// TwinCAT 3 PLC project PLC1
// ProgramVersion: 3.1.4026.21
// libraries:
//   Tc2_Standard, * (Beckhoff Automation GmbH)
//   Tc2_System, * (Beckhoff Automation GmbH)
//   Tc2_TcpIp, * (Beckhoff Automation GmbH)
//   Tc2_Utilities, * (Beckhoff Automation GmbH)
// project tree:
//   DUTs/ESP/ EspPacketTerminater.TcDUT (not stored), EspPacketHeader.TcDUT, UpdaterEntry.TcDUT
//   DUTs/RtUdp/ IpAdrUnion.TcDUT (not stored)
//   Functions/ BytesToIpv4.TcPOU (not stored), BytesToUint.TcPOU, BytesToUlint.TcPOU (not stored), CalculatePowerConsumption.TcPOU (not stored), HeaderEndianSwap.TcPOU, Ipv4ToBytes.TcPOU, TailEndianSwap.TcPOU (not stored)
//   GVLs/ GVL_Udp.TcGVL (not stored)
//   Interfaces/ ITF_Cyclic.TcIO (not stored), ITF_EspHost.TcIO, ITF_Node.TcIO, ITF_LinkedList.TcIO (not stored), ITF_NodeFactory.TcIO, ITF_UdpConnection.TcIO, ITF_Updater.TcIO, ITF_UpdaterRegistry.TcIO
//   Object/ESP/ EspHost.TcPOU, UpdaterRegistry.TcPOU, Updater_TestPacket.TcPOU
//   Object/Factories/ EspHostFactory.TcPOU (not stored)
//   Object/IO/ RgbController.TcPOU (not stored)
//   Object/Linked List/ List.TcPOU (not stored)
//   Object/UDP/ DataDecoder.TcPOU, UdpRealtimeSocket.TcPOU, UdpWindowsSocket.TcPOU
//   POUs/ Application.TcPOU, EnergyCalculator.TcPOU, MAIN.TcPOU, MessageBuffer.TcPOU, Tests.TcPOU (not stored), Utility.TcPOU
//   Tasks/ Task_4.TcTTO, _aux.TcTTO (not stored)
//   Tests/ EspNodeController.TcPOU (not stored), GVL_Test.TcGVL, TestHarness.TcPOU (not stored), TestNode.TcPOU, TestNodeFactory.TcPOU, Tests_ListAndFactory.TcPOU, Tests_Udp.TcPOU
// real-time tasks:
//   TASK Task 4: cycle T#100us, priority 1, ADS port 350
//   TASK Aux: cycle T#10ms, priority 2, ADS port 351
// I/O:
//   DEVICE Wifi Router
//   DEVICE Rail IO, AmsNetId 5.143.167.204.4.1
//     Term 1 (EK1200) [EK1200-5000 EtherCAT Power supply (2A E-Bus)]
//       Term 2 (EL9227-5500) [EL9227-5500 Overcurrent protection 24V DC, 2Ch., max. 10A (sum), adjustable, extended functionalities]
//       Term 3 (EL2088) [EL2088 8Ch. Dig. Output 24V, 0.5A, switching to negative]
//       Term 4 (EL9011) [EL9011 End Terminal]
// variable links:
//   PLC1/PLC1 Instance <-> Rail IO/Term 1 (EK1200)/Term 2 (EL9227-5500)
//     Aux Inputs/Utility.EL9227Ch2.MDP5001_922_Input/MDP5001_922_Current <-> OCP Inputs Channel 2/Current
//     Aux Inputs/Utility.EL9227Ch2.MDP5001_922_Input/MDP5001_922_Load <-> OCP Inputs Channel 2/Load
//     Aux Inputs/Utility.EL9227Ch2.MDP5001_922_Input/MDP5001_922_Status <-> OCP Inputs Channel 2/Status
//     Aux Inputs/Utility.EL9227Ch2.MDP5001_922_Input/MDP5001_922_Voltage_In <-> OCP Inputs Channel 2/Voltage In
//     Aux Inputs/Utility.EL9227Ch2.MDP5001_922_Input/MDP5001_922_Voltage_Out <-> OCP Inputs Channel 2/Voltage Out
//     Aux Outputs/Utility.EL9227Ch2.MDP5001_922_Output/MDP5001_922_Control <-> OCP Outputs Channel 2/Control
//     Task_4 Inputs/Utility.EL9227Ch1.MDP5001_922_Input/MDP5001_922_Current <-> OCP Inputs Channel 1/Current
//     Task_4 Inputs/Utility.EL9227Ch1.MDP5001_922_Input/MDP5001_922_Load <-> OCP Inputs Channel 1/Load
//     Task_4 Inputs/Utility.EL9227Ch1.MDP5001_922_Input/MDP5001_922_Status <-> OCP Inputs Channel 1/Status
//     Task_4 Inputs/Utility.EL9227Ch1.MDP5001_922_Input/MDP5001_922_Voltage_In <-> OCP Inputs Channel 1/Voltage In
//     Task_4 Inputs/Utility.EL9227Ch1.MDP5001_922_Input/MDP5001_922_Voltage_Out <-> OCP Inputs Channel 1/Voltage Out
//     Task_4 Outputs/Utility.EL9227Ch1.MDP5001_922_Output/MDP5001_922_Control <-> OCP Outputs Channel 1/Control
//   PLC1/PLC1 Instance <-> Rail IO/Term 1 (EK1200)/Term 3 (EL2088)
//     Task_4 Outputs/Utility.LedStrip._Blue <-> Channel 5/Output
//     Task_4 Outputs/Utility.LedStrip._Green <-> Channel 3/Output
//     Task_4 Outputs/Utility.LedStrip._Red <-> Channel 1/Output

CONFIGURATION PLC1
    RESOURCE PLC ON TwinCAT3
        TASK Task_4(INTERVAL := T#200us, PRIORITY := 1);
        PROGRAM MAIN WITH Task_4 : MAIN;
    END_RESOURCE
END_CONFIGURATION

// ---- DUTs/ESP/EspPacketHeader.TcDUT
TYPE EspPacketHeader :
STRUCT
	StartDelimiter			: UINT := 693;
	PayloadSize				: UINT;
	Reserved1				: ARRAY [1..4] OF BYTE;
	SlaveUid				: ULINT;
	MessageCounter			: ULINT;
	SendersTimestamp		: ULINT;
	TimeDifference			: UDINT;
	NumberOfChainedSLaves	: BYTE;
	EspType					: BYTE;
	Flags					: BYTE;
	HeaderVersion			: BYTE;
	NetworkId				: BYTE;
	ChainDistance			: BYTE;
	JumpsToLive				: BYTE;
	Reserved2				: BYTE;
	CRC32					: UDINT;
END_STRUCT
END_TYPE

// ---- DUTs/ESP/UpdaterEntry.TcDUT
TYPE UpdaterEntry :
STRUCT
	TypeID	: BYTE;
	Version	: BYTE;
	Updater	: ITF_Updater;
END_STRUCT
END_TYPE

// ---- Tests/GVL_Test.TcGVL
{attribute 'qualified_only'}
VAR_GLOBAL
	
END_VAR

// ---- Interfaces/ITF_EspHost.TcIO
INTERFACE ITF_EspHost

METHOD CyclicUpdate : BOOL
VAR_INPUT
END_VAR
END_METHOD

METHOD GetDataBuffer : BOOL
VAR_INPUT
	Address	: REFERENCE TO PVOID;
	Size	: REFERENCE TO UDINT;
END_VAR
END_METHOD

METHOD GetMetadata : EspPacketHeader
VAR_INPUT
END_VAR
END_METHOD

METHOD GetPacketToSend : BOOL
VAR_INPUT
	Address	: REFERENCE TO PVOID;
	Size	: REFERENCE TO UDINT;
END_VAR
END_METHOD

METHOD SetEspType : BOOL
VAR_INPUT
	EspType	: BYTE;
END_VAR
END_METHOD

METHOD SetUID : BOOL
VAR_INPUT
	UID	: ULINT;
END_VAR
END_METHOD

METHOD UpdateMetadata : BOOL
VAR_INPUT
	Data	: EspPacketHeader;
END_VAR
END_METHOD

END_INTERFACE

// ---- Interfaces/ITF_Node.TcIO
INTERFACE ITF_Node

METHOD GetLastNode : ITF_Node
VAR_INPUT
END_VAR
END_METHOD

METHOD GetMyPointer : PVOID
END_METHOD

METHOD GetNextNode : ITF_Node
VAR_INPUT
END_VAR
END_METHOD

METHOD GetPositionInList : UINT
VAR_INPUT
END_VAR
END_METHOD

METHOD SetLastNode : BOOL
VAR_INPUT
	Node	: ITF_Node;
END_VAR
END_METHOD

METHOD SetNextNode : BOOL
VAR_INPUT
	Node	: ITF_Node;
END_VAR
END_METHOD

METHOD SetPositionInList : BOOL
VAR_INPUT
	Index		: UINT;
END_VAR
END_METHOD

END_INTERFACE

// ---- Interfaces/ITF_NodeFactory.TcIO
INTERFACE ITF_NodeFactory

METHOD CreateNode : ITF_Node
VAR_INPUT
END_VAR
END_METHOD

METHOD DestroyNode : BOOL
VAR_INPUT
	Ptr		: PVOID;
END_VAR
END_METHOD

METHOD DoesCreateEqualDestroy : BOOL
END_METHOD

END_INTERFACE

// ---- Interfaces/ITF_UdpConnection.TcIO
INTERFACE ITF_UdpConnection EXTENDS ITF_Cyclic

METHOD IsConnected : BOOL
VAR_INPUT
END_VAR
END_METHOD

METHOD IsSending : BOOL
VAR_INPUT
END_VAR
END_METHOD

PROPERTY LastReceivedIp : T_IPv4Addr
GET
END_GET
END_PROPERTY

PROPERTY ReceiveBufferReference : REFERENCE TO ARRAY [0..TCPADS_MAXUDP_BUFFSIZE - 1] OF BYTE;
GET
END_GET
END_PROPERTY

METHOD TryCloseConnection : HRESULT
VAR_INPUT
END_VAR
END_METHOD

METHOD TryOpenConnection : HRESULT
VAR_INPUT
END_VAR
END_METHOD

METHOD TryReadReceiveBuffer : HRESULT
VAR_INPUT
	DataBuffer		: REFERENCE TO ARRAY [0..TCPADS_MAXUDP_BUFFSIZE - 1] OF BYTE;
END_VAR
END_METHOD

METHOD TrySendData : HRESULT
VAR_INPUT
	IpAddress		: T_IPv4Addr;
	Port			: UDINT;
	DataAddress		: PVOID;
	DataLength		: UDINT;
END_VAR
END_METHOD

END_INTERFACE

// ---- Interfaces/ITF_Updater.TcIO
INTERFACE ITF_Updater

METHOD GetTypeID : BYTE
VAR_INPUT
END_VAR
END_METHOD

METHOD GetVersion : BYTE
VAR_INPUT
END_VAR
END_METHOD

METHOD TryApplyPayload : HRESULT
VAR_INPUT
	PacketAddress	: PVOID;
	PacketLength	: UINT;
	EspHost			: ITF_EspHost;
END_VAR
END_METHOD

METHOD TryGetContents : HRESULT
VAR_INPUT
	Host	: ITF_EspHost;
	Content	: REFERENCE TO STRING(1024);
END_VAR
END_METHOD

METHOD TrySendInstruction : HRESULT
VAR_INPUT
END_VAR
END_METHOD

END_INTERFACE

// ---- Interfaces/ITF_UpdaterRegistry.TcIO
INTERFACE ITF_UpdaterRegistry

METHOD Reset : BOOL
VAR_INPUT
END_VAR
END_METHOD

METHOD ResolveUpdater : ITF_Updater
VAR_INPUT
	TypeID	: BYTE;
	Version	: BYTE;
END_VAR
END_METHOD

METHOD TryRegister : HRESULT
VAR_INPUT
	Updater	: ITF_Updater;
END_VAR
END_METHOD

END_INTERFACE

// ---- POUs/MAIN.TcPOU
PROGRAM MAIN
VAR
	Test	: BOOL := FALSE;
	i		: INT;
END_VAR


i := i + 1;


IF Test THEN
	
	Tests();
	
ELSE
	
	Application();
	
END_IF

END_PROGRAM

// ---- POUs/Application.TcPOU
PROGRAM Application
VAR CONSTANT
	Port 					: UDINT := 10050;
END_VAR
VAR
	UdpWin10				: UdpWindowsSocket('192.168.137.1', Port);
	UdpRt					: UdpRealtimeSocket(Port);
	Udp						: ITF_UdpConnection := UdpRt;
	
	EspFactory				: EspHostFactory;
	List					: List(EspFactory);
	
	DataDecoder				: DataDecoder(Udp, List);
	UpdaterRegistry			: UpdaterRegistry;
	TestUpdater				: Updater_TestPacket;
	
	Init					: BOOL := FALSE;
	i						: BYTE;
	j						: UINT;
	State					: BYTE;
	hr						: HRESULT;

	ReceivedIP				: T_IPv4Addr;
	InputHeader				: EspPacketHeader;	
	TempEspPtr				: POINTER TO EspHost;
	TempEsp					: ITF_EspHost;
	TempEspHeader			: EspPacketHeader;
	
	PacketToSendAdr			: PVOID;
	PacketToSendLength		: UDINT;
	
	ReceivedPacketType		: BYTE;
	ReceivedPacketAddress	: PVOID;
	ReceivedPacketLength	: UINT;
	ReceivedDataLength		: UINT;
	
	PacketsProcessed		: ULINT;
END_VAR


IF NOT Init THEN

	IF Udp.TryOpenConnection() <> S_OK THEN
		
		RETURN;
	
	END_IF

	UpdaterRegistry.TryRegister(TestUpdater);
	
	Init := TRUE;

END_IF





// Multiple processing calls per cycle are possible

FOR i := 0 TO 9 BY 1 DO
	
	Udp.CyclicUpdate();
	
	CASE State OF
		
		0:	// Is data available
			
			hr := DataDecoder.TryFindPacketInBuffer(ReceivedPacketType, ReceivedPacketAddress, ReceivedPacketLength, ReceivedDataLength);
			
			IF hr = S_OK THEN
				
				ReceivedIP := UdpRt.LastReceivedIp;
				
				State := 1;
				
			ELSIF hr <> S_PENDING THEN
				
				EXIT;
				
			END_IF
			
	

		1:	// Decode header
		
			InputHeader := DataDecoder.GetPacketHeader();

			IF InputHeader.SlaveUid = 0 THEN
				
				// Clear buffer
				
				State := 0;
				
			END_IF
			
			State := 2;



		2:	// Check CRC
		
			// CRC Check Function on TargetHeader
			
			// If fail, clear buffer, state := 0
			
			State := 3;



		3:	// Find UID in list
		
			IF List.GetListLength() = 0 THEN
				
				State := 4;
				
			END_IF
		
			FOR j := 1 TO List.GetListLength() BY 1 DO
			
				TempEspPtr := List.GetNode(j).GetMyPointer();
				
				IF TempEspPtr = 0 THEN
					
					// No matching device in list, create
					
					State := 4;
					
				ELSE
					
					// Check if correct UID
					
					TempEsp := TempEspPtr^;
				
					TempEspHeader := TempEsp.GetMetadata();
					
					IF InputHeader.SlaveUid = TempEspHeader.SlaveUid THEN
						
						State := 5;
						
						EXIT;
						
					END_IF
					
				END_IF
				
			END_FOR	
			
			IF j = List.GetListLength() + 1 THEN
				
				State := 4;
				
			END_IF
			
			
			
		4:	// Create device in list
			
			IF List.CreateNode() THEN
						
				TempEspPtr := List.GetNode(List.GetListLength()).GetMyPointer();
				
				TempEsp := TempEspPtr^;
				
				TempEsp.SetUID(InputHeader.SlaveUid);
				
				TempEsp.SetEspType(ReceivedPacketType);
				
				State := 5;
			
			END_IF
			
			
			
		5:	// Apply data
		
			IF TempEsp.UpdateMetadata(InputHeader) THEN
				
				IF TempEsp.GetPacketToSend(PacketToSendAdr, PacketToSendLength) THEN
					
					TempEsp.CyclicUpdate();
					
					State := 6;

				ELSE
					
					State := 7;
	
				END_IF
				
			END_IF
		
		
		
		6:	// Send data
		
			hr := UdpRt.TrySendData(ReceivedIP, Port, PacketToSendAdr, PacketToSendLength);
			
			IF hr <> S_PENDING AND SUCCEEDED(hr) THEN
				
				State := 7;
				
			ELSIF FAILED(hr) THEN
				
				State := 8;
				
			END_IF
		
		
		
		7:	// System function OK
			
			ReceivedIP := '';
			MEMSET(ADR(InputHeader), 0, 48);
			TempEspPtr := 0;
			TempEsp := 0;
			MEMSET(ADR(TempEspHeader), 0, 48);
			DataDecoder.ClearBufferAtLocation(ReceivedPacketAddress, ReceivedPacketLength);
			
			PacketsProcessed := PacketsProcessed + 1;
			State := 0;
			
			
		
		
		8:	// System RX OK, TX FAIL
		
// 		
// 		
// 		
// 		5:
// 		
// 			hr := TempUpdater.TryApplyPayload(ReceivedPacketAddress, ReceivedPacketLength, TempEsp);
// 			
// 			IF hr <> S_PENDING AND SUCCEEDED(hr) THEN
// 				
// 				TempEsp.UpdateMetadata(DataDecoder.CreateMetadataUpdate());
// 				
// 				DataDecoder.ClearBufferAtLocation(ReceivedPacketAddress, ReceivedPacketLength);
// 				
// 				ReceivedPacketAddress := 0;
// 				ReceivedPacketLength := 0;
// 				ReceivedPacketType := 0;
// 			
// 				TargetEspUID := 0;
// 				TempEspPtr := 0;	
// 				TempEsp := 0;
// 				MEMSET(ADR(TempEspHeader), 0, SIZEOF(TempEspHeader));
// 				TempUpdater := 0;
// 				
// 				State := 0;
// 				
// 			END_IF
// 		
// 		
// 			
// 			
// 		1:
// 		
// 			TempUpdater := UpdaterRegistry.ResolveUpdater(ReceivedPacketType, 1);
// 			
// 			IF TempUpdater = 0 THEN
// 				
// 				;// ERROR
// 				
// 			END_IF
// 			
// 			State := 2;
// 			
// 		
// 		
// 		2:
// 		
// 			TargetEspUID := DataDecoder.GetPacketUID();
// 			
// 			IF TargetEspUID = 0 THEN
// 				
// 				;// ERROR
// 				
// 			END_IF
// 			
// 			State := 3;
// 			
// 			
// 			
// 		3:
// 		
// 			FOR j := 1 TO List.GetListLength() BY 1 DO
// 			
// 				TempEspPtr := List.GetNode(j).GetMyPointer();
// 			
// 				TempEsp := TempEspPtr^;
// 				
// 				TempEspHeader := TempEsp.GetMetadata();
// 				
// 				IF TargetEspUID = TempEspHeader.SlaveUid THEN
// 					
// 					FoundEsp := TRUE;
// 					
// 					EXIT;
// 					
// 				END_IF
// 				
// 			END_FOR
// 			
// 			IF FoundEsp THEN
// 				
// 				FoundEsp := FALSE;
// 				
// 				State := 5;
// 				
// 			ELSE
// 				
// 				State := 4;
// 				
// 			END_IF
// 			
// 			
// 			
// 		4:
// 			
// 			IF List.CreateNode() THEN
// 						
// 				TempEspPtr := List.GetNode(List.GetListLength()).GetMyPointer();
// 				
// 				TempEsp := TempEspPtr^;
// 				
// 				TempEsp.SetUID(TargetEspUID);
// 				
// 				TempEsp.SetEspType(ReceivedPacketType);
// 				
// 				State := 5;
// 			
// 			END_IF
// 		
// 		
// 		
// 		5:
// 		
// 			hr := TempUpdater.TryApplyPayload(ReceivedPacketAddress, ReceivedPacketLength, TempEsp);
// 			
// 			IF hr <> S_PENDING AND SUCCEEDED(hr) THEN
// 				
// 				TempEsp.UpdateMetadata(DataDecoder.CreateMetadataUpdate());
// 				
// 				DataDecoder.ClearBufferAtLocation(ReceivedPacketAddress, ReceivedPacketLength);
// 				
// 				ReceivedPacketAddress := 0;
// 				ReceivedPacketLength := 0;
// 				ReceivedPacketType := 0;
// 			
// 				TargetEspUID := 0;
// 				TempEspPtr := 0;	
// 				TempEsp := 0;
// 				MEMSET(ADR(TempEspHeader), 0, SIZEOF(TempEspHeader));
// 				TempUpdater := 0;
// 				
// 				State := 0;
// 				
// 			END_IF
			
	END_CASE

END_FOR

END_PROGRAM

// ---- Object/UDP/UdpWindowsSocket.TcPOU
FUNCTION_BLOCK UdpWindowsSocket IMPLEMENTS ITF_UdpConnection
VAR
	IpAddress			: T_IPv4Addr;
	Port				: UDINT;
	ReceiveBuffer		: ARRAY [0..TCPADS_MAXUDP_BUFFSIZE - 1] OF BYTE;
	
	OpenSocket			: FB_SocketUdpCreate;
	Receive				: FB_SocketUdpReceiveFrom;
	Send				: FB_SocketUdpSendTo;
	SendState			: BYTE;
	Sending 			: BOOL;
	PacketsSent			: ULINT;
	CloseSocket			: FB_SocketClose;
	
	IsConnectionOpen	: BOOL;
END_VAR

METHOD CyclicUpdate : BOOL
VAR
	i	: BYTE;
END_VAR
OpenSocket
(
	sSrvNetId 	:= '', 
	sLocalHost	:= IpAddress, 
	nLocalPort	:= Port, 
);

Send
(
	sSrvNetId	:= '', 
	hSocket		:= OpenSocket.hSocket, 
);

FOR i := 0 TO 9 BY 1 DO
	
	Receive
	(
		sSrvNetId	:= '', 
		hSocket		:= OpenSocket.hSocket, 
		cbLen		:= SIZEOF(ReceiveBuffer), 
		pDest		:= ADR(ReceiveBuffer) 
	);
	
	IF IsSending() OR NOT IsConnectionOpen THEN
	
		Receive(bExecute := FALSE);
		
	ELSE
		
		Receive(bExecute := NOT(Receive.bExecute));
	
	END_IF

END_FOR


CloseSocket
(
	sSrvNetId	:= '', 
	hSocket		:= OpenSocket.hSocket, 
);

IF OpenSocket.hSocket.handle <> 0 AND OpenSocket.bExecute THEN
	
	IsConnectionOpen := TRUE;
	
ELSE

	IsConnectionOpen := FALSE;

END_IF
END_METHOD

//FB_Exit must be implemented explicitly. If there is an implementation, then the
//method is called before the controller removes the code of the function block instance
//(implicit call). The return value is not evaluated.
METHOD FB_Exit: BOOL
VAR_INPUT
    bInCopyCode: BOOL;  // TRUE: the exit method is called in order to leave the instance which will be copied afterwards (online change).  
END_VAR
TryCloseConnection();
END_METHOD

//FB_Init is always available implicitly and it is used primarily for initialization.
//The return value is not evaluated. For a specific influence, you can also declare the
//methods explicitly and provide additional code there with the standard initialization
//code. You can evaluate the return value.
METHOD FB_Init: BOOL
VAR_INPUT
    bInitRetains: BOOL; // TRUE: the retain variables are initialized (reset warm / reset cold)
    bInCopyCode: BOOL;  // TRUE: the instance will be copied to the copy code afterward (online change) 
	IpAddress	: T_IPv4Addr;
	Port		: UDINT;  
END_VAR
THIS^.IpAddress := IpAddress;
THIS^.Port := Port;
END_METHOD

METHOD IsConnected : BOOL
IsConnected := IsConnectionOpen;

RETURN;
END_METHOD

METHOD IsSending : BOOL
IsSending := Sending;

RETURN;
END_METHOD

{warning 'Add property implementation'}
PROPERTY LastReceivedIp : T_IPv4Addr
GET
LastReceivedIp := Receive.sRemoteHost;
END_GET
END_PROPERTY

{warning 'Add property implementation'}
PROPERTY LastReceivedPort : UDINT
GET
LastReceivedPort := Receive.nRemotePort;
END_GET
END_PROPERTY

{warning 'Add property implementation'}
PROPERTY ReceiveBufferReference : REFERENCE TO ARRAY [0..(TCPADS_MAXUDP_BUFFSIZE - 1)] OF BYTE
GET
ReceiveBufferReference REF= ReceiveBuffer;
END_GET
END_PROPERTY

METHOD TryCloseConnection : HRESULT
TryCloseConnection := S_PENDING;

OpenSocket(bExecute := FALSE);

CloseSocket(bExecute := TRUE);

IF OpenSocket.hSocket.handle = 0 THEN
	
	TryCloseConnection := S_OK;

ELSIF OpenSocket.bError THEN

	TryCloseConnection := -1;	

END_IF

RETURN;
END_METHOD

METHOD TryOpenConnection : HRESULT
TryOpenConnection := S_PENDING;

CloseSocket(bExecute := FALSE);

OpenSocket(bExecute := TRUE);

IF OpenSocket.hSocket.handle <> 0 THEN
	
	TryOpenConnection := S_OK;

ELSIF OpenSocket.bError THEN

	TryOpenConnection := -1;	

END_IF

RETURN;
END_METHOD

METHOD TryReadReceiveBuffer : HRESULT
VAR_INPUT
	DataBuffer		: REFERENCE TO ARRAY [0..TCPADS_MAXUDP_BUFFSIZE - 1] OF BYTE;
END_VAR
VAR
	i				: UDINT;
END_VAR
TryReadReceiveBuffer := S_PENDING;

IF ReceiveBuffer[0] = 0 THEN
	
	TryReadReceiveBuffer := -1;

	RETURN;	

END_IF

FOR i := 0 TO TCPADS_MAXUDP_BUFFSIZE BY 1 DO
	
	IF ReceiveBuffer[i] = 0 THEN
		
		EXIT;
		
	END_IF

	DataBuffer[i] := ReceiveBuffer[i];

END_FOR

IF ReceiveBuffer[0] <> 0 THEN
	
	TryReadReceiveBuffer := S_OK;

ELSE

	TryReadReceiveBuffer := -2;

END_IF

RETURN;
END_METHOD

METHOD TrySendData : HRESULT
VAR_INPUT
	IpAddress		: T_IPv4Addr;
	Port			: UDINT;
	DataAddress		: PVOID;
	DataLength		: UDINT;
END_VAR
TrySendData := S_PENDING;

IF NOT IsConnected() THEN
	
	TrySendData := -1;
	
	RETURN;

END_IF

Send
(
	sRemoteHost	:= IpAddress, 
	nRemotePort	:= Port, 
	cbLen		:= DataLength, 
	pSrc		:= DataAddress, 
	bExecute	:= TRUE, 
);

Sending := TRUE;

CASE SendState OF
	
	0:
	
		IF Send.bBusy THEN
			
			SendState := 1;
			
		END_IF



	1:
	
		IF Send.bError THEN
			
			Send(bExecute := FALSE);
			
			TrySendData := -1;
			
			SendState := 0;
			
			Sending := FALSE;
			
			RETURN;
		
		ELSIF NOT Send.bBusy THEN
			
			Send(bExecute := FALSE);
		
			TrySendData := S_OK;
			
			PacketsSent := PacketsSent + 1;
			
			SendState := 0;
			
			Sending := FALSE;
			
			RETURN;
		
		END_IF
END_CASE
END_METHOD

END_FUNCTION_BLOCK

// ---- Object/UDP/UdpRealtimeSocket.TcPOU
{attribute 'c++_compatible'}
FUNCTION_BLOCK UdpRealtimeSocket IMPLEMENTS ITcIoUdpProtocolRecv, ITF_UdpConnection
VAR
	{attribute 'TcInitSymbol'}
	_ObjectId				: OTCID; 
	_ipUdp					: ITcIoUdpProtocol;
	_UdpPort				: UINT := 10000;
	_ReceivedPackets		: ULINT;
	_LastReceivedIpAddr 	: IpAdrUnion;
	_LastReceivedPort		: UDINT; 
	_LastSentIpAddr			: IpAdrUnion;
	_hrInit 				: HRESULT;
	_SocketOpen				: BOOL;
	_Sending				: BOOL;
	
	_ReceivedData			: PVOID;
	_ReceivedDataLength		: UDINT;
		
	_ReceiveBuffer			: ARRAY [0..TCPADS_MAXUDP_BUFFSIZE - 1] OF BYTE;

END_VAR

METHOD CyclicUpdate : BOOL
IF _ipUdp <> 0 THEN
	
	_ipUdp.CheckReceived();
	
END_IF

IF _ReceivedData <> 0 THEN

	MEMCPY(ADR(_ReceiveBuffer), _ReceivedData, _ReceivedDataLength);
	
	_ReceivedData := 0;
	
	_ReceivedDataLength := 0;

END_IF
END_METHOD

METHOD FB_exit : BOOL
VAR_INPUT
	bInCopyCode : BOOL; // if TRUE, the exit method is called for exiting an instance that is copied afterwards (online change).
END_VAR
IF (NOT bInCopyCode AND _ipUdp <> 0) THEN //Shutdown
	_ipUdp.UnregisterReceiver(_UdpPort);
	FW_SafeRelease(ADR(_ipUdp));
	_SocketOpen := FALSE;
	FB_exit := TRUE;
ELSE
	FB_exit := FALSE;
END_IF
END_METHOD

METHOD FB_init : BOOL
VAR_INPUT
	bInitRetains : BOOL; // if TRUE, the retain variables are initialized (warm start / cold start)
	bInCopyCode : BOOL;  // if TRUE, the instance afterwards gets moved into the copy code (online change)
	Port	: UDINT;
END_VAR
VAR
	//ipSrv: ITComObjectServer;
END_VAR
_UdpPort := TO_UINT(Port);
// 
// IF NOT bInCopyCode THEN // no online change
// 	IF ipUdp = 0 AND ObjectId <> 0 THEN
// 	 hrInit := FW_ObjMgr_GetObjectInstance(oid:=ObjectId, iid:=TC_GLOBAL_IID_LIST.IID_ITcIoUdpProtocol, pipUnk:=ADR(ipUdp) );
// 		IF SUCCEEDED(hrInit) THEN 
// 			IF SUCCEEDED(ipUdp.RegisterReceiver(UdpPort, THIS^)) THEN //open port
// 				SocketOpen := TRUE;
// 				FB_init := TRUE;
// 			ELSE 
// 				FB_init := FALSE; 
// 				FW_SafeRelease(ADR(ipUdp));
// 			END_IF
// 		END_IF
// 	ELSIF ObjectId = 0 THEN 
// 		FB_init := FALSE; 
// 		hrInit := ERR_INVALID_PARAM; 				
// 	END_IF
// END_IF
END_METHOD

METHOD FB_reinit : BOOL
VAR_INPUT
END_VAR
IF (_ipUdp <> 0) THEN 
  _ipUdp.RegisterReceiver(_UdpPort, THIS^);
  _SocketOpen := TRUE;
  FB_reinit := TRUE; 
END_IF
END_METHOD

METHOD IsConnected : BOOL
IsConnected := _SocketOpen;

RETURN;
END_METHOD

METHOD IsSending : BOOL
IsSending := _Sending;

RETURN;
END_METHOD

PROPERTY LastReceivedIp : T_IPv4Addr
GET
LastReceivedIp := BytesToIpv4(_LastReceivedIpAddr.IpByte);
END_GET
END_PROPERTY

{warning 'Add property implementation'}
PROPERTY LastReceivedPort : UDINT
GET
LastReceivedPort := _LastReceivedPort;
END_GET
END_PROPERTY

{warning 'Add property implementation'}
PROPERTY ReceiveBufferReference : REFERENCE TO ARRAY [0..(TCPADS_MAXUDP_BUFFSIZE - 1)] OF BYTE
GET
ReceiveBufferReference REF= _ReceiveBuffer;
END_GET
END_PROPERTY

{attribute 'object_name' := 'ReceiveData'}
{attribute 'c++_compatible'}
{attribute 'pack_mode' := '4'}
{attribute 'show'}
{attribute 'minimal_input_size' := '4'}
METHOD ReceiveData : HRESULT
VAR_INPUT
	ipAddr	: UDINT;
	udpDestPort	: UINT;
	udpSrcPort	: UINT;
	nData	: UDINT;
	pData	: PVOID;
	pVlan	: POINTER TO ETYPE_VLAN_HEADER := 0;
END_VAR
_ReceivedPackets := _ReceivedPackets + 1;

_LastReceivedIpAddr.IpUdint := ipAddr;

_LastReceivedPort := TO_UDINT(udpDestPort);

IF _ipUdp <> 0 THEN
	
	//ipUdp.SendData(ipAddr, udpSrcPort, udpDestPort, nData, pData, TRUE, 0); // send data back

	_ReceivedData := pData;
	
	_ReceivedDataLength := nData;
	
END_IF
END_METHOD

{attribute 'object_name' := 'TcAddRef'}
{attribute 'c++_compatible'}
{attribute 'pack_mode' := '4'}
{attribute 'show'}
{attribute 'minimal_input_size' := '4'}
METHOD TcAddRef : UDINT
END_METHOD

{attribute 'object_name' := 'TcQueryInterface'}
{attribute 'c++_compatible'}
{attribute 'pack_mode' := '4'}
{attribute 'show'}
{attribute 'minimal_input_size' := '4'}
METHOD TcQueryInterface : HRESULT
VAR_INPUT
	iid	: REFERENCE TO IID;
	pipItf	: POINTER TO PVOID;
END_VAR
VAR
   ipUdpRecv : ITcIoUdpProtocolRecv;
   ipUnknown : ITcUnknown;   
END_VAR
IF GuidsEqual(ADR(iid), ADR(TC_GLOBAL_IID_LIST.IID_ITcIoUdpProtocolRecv)) THEN
   ipUdpRecv := THIS^; // cast to interface pointer
   pipItf^ := ITCUNKNOWN_TO_PVOID(ipUdpRecv);
   TcAddRef();
   TcQueryInterface := S_OK;
ELSIF GuidsEqual(ADR(iid), ADR(TC_GLOBAL_IID_LIST.IID_ITcUnknown)) THEN
   ipUnknown := THIS^; // cast to interface pointer
   pipItf^ := ITCUNKNOWN_TO_PVOID(ipUnknown);
   TcAddRef();
   TcQueryInterface := S_OK;
ELSE
   TcQueryInterface := E_HRESULTAdsErr.NOINTERFACE ; //Call super if this fb extends some other
END_IF
END_METHOD

{attribute 'object_name' := 'TcRelease'}
{attribute 'c++_compatible'}
{attribute 'pack_mode' := '4'}
{attribute 'show'}
{attribute 'minimal_input_size' := '4'}
METHOD TcRelease : UDINT
END_METHOD

METHOD TryCloseConnection : HRESULT
TryCloseConnection := S_PENDING;

IF (_ipUdp <> 0) THEN //Shutdown
	_ipUdp.UnregisterReceiver(_UdpPort);
	FW_SafeRelease(ADR(_ipUdp));
	_SocketOpen := FALSE;
	TryCloseConnection := S_OK;
ELSE
	TryCloseConnection := S_FALSE;
END_IF
END_METHOD

METHOD TryOpenConnection : HRESULT
TryOpenConnection := S_PENDING;

IF IsConnected() THEN
	
	TryOpenConnection := S_OK;
	
ELSIF _ipUdp = 0 AND _ObjectId <> 0 THEN
 	_hrInit := FW_ObjMgr_GetObjectInstance(oid:=_ObjectId, iid:=TC_GLOBAL_IID_LIST.IID_ITcIoUdpProtocol, pipUnk:=ADR(_ipUdp) );
	IF SUCCEEDED(_hrInit) THEN 
		IF SUCCEEDED(_ipUdp.RegisterReceiver(_UdpPort, THIS^)) THEN //open port
			_SocketOpen := TRUE;
			TryOpenConnection := S_OK;
		ELSE 
			TryOpenConnection := -1; 
			FW_SafeRelease(ADR(_ipUdp));
		END_IF
	END_IF
ELSIF _ObjectId = 0 THEN 
	TryOpenConnection := -2; 
	_hrInit := ERR_INVALID_PARAM; 				
END_IF

RETURN;
END_METHOD

METHOD TryReadReceiveBuffer : HRESULT
VAR_INPUT
	DataBuffer		: REFERENCE TO ARRAY [0..TCPADS_MAXUDP_BUFFSIZE - 1] OF BYTE;
END_VAR
VAR
	i				: UDINT;
END_VAR
TryReadReceiveBuffer := S_PENDING;

IF _ReceiveBuffer[0] = 0 THEN
	
	TryReadReceiveBuffer := -1;

	RETURN;	

END_IF

FOR i := 0 TO TCPADS_MAXUDP_BUFFSIZE BY 1 DO
	
	IF _ReceiveBuffer[i] = 0 THEN
		
		EXIT;
		
	END_IF

	DataBuffer[i] := _ReceiveBuffer[i];

END_FOR

IF _ReceiveBuffer[0] <> 0 THEN
	
	TryReadReceiveBuffer := S_OK;

ELSE

	TryReadReceiveBuffer := -2;

END_IF

RETURN;
END_METHOD

METHOD TrySendData : HRESULT
VAR_INPUT
	IpAddress	: T_IPv4Addr;
	Port		: UDINT;
	DataAddress	: PVOID;
	DataLength	: UDINT;
END_VAR
VAR
	hr	: HRESULT;
END_VAR
TrySendData := S_PENDING;

IF NOT IsConnected() THEN
	
	TrySendData := -1;
	
	RETURN;

END_IF

hr := S_PENDING;

_LastSentIpAddr.IpByte := Ipv4ToBytes(IpAddress);

hr := _ipUdp.SendData(_LastSentIpAddr.IpUdint, _UdpPort, TO_UINT(Port), DataLength, DataAddress, TRUE, 0);

IF hr <> S_PENDING AND SUCCEEDED(hr) THEN
	
	TrySendData := S_OK;
	
ELSIF FAILED(hr) THEN
	
	TrySendData := -1;	

END_IF
END_METHOD

END_FUNCTION_BLOCK

// ---- Functions/Ipv4ToBytes.TcPOU
FUNCTION Ipv4ToBytes : ARRAY [0..3] OF BYTE
VAR_INPUT
    IpAddress : T_IPv4Addr;
END_VAR
VAR
    i 		: BYTE := 0;
	j		: BYTE := 1;
	t1		: STRING;
	t2		: STRING;
	t3		: STRING;
	t4		: STRING;
END_VAR


FOR i := 0 TO 16 BY 1 DO
	
	IF IpAddress[i] = 0 THEN
		
		EXIT;
		
	ELSIF IpAddress[i] = 46 THEN // 46 = '.'
		
		j := j + 1;
		
	ELSE

		CASE j OF
			
			1:
				t1 := CONCAT(t1, F_ToCHR(IpAddress[i]));
			
			2:
				t2 := CONCAT(t2, F_ToCHR(IpAddress[i]));
				
			3:
				t3 := CONCAT(t3, F_ToCHR(IpAddress[i]));
				
			4:
				t4 := CONCAT(t4, F_ToCHR(IpAddress[i]));
			
		END_CASE
	
	END_IF
	
END_FOR

Ipv4ToBytes[0] := STRING_TO_BYTE(t4);

Ipv4ToBytes[1] := STRING_TO_BYTE(t3);

Ipv4ToBytes[2] := STRING_TO_BYTE(t2);

Ipv4ToBytes[3] := STRING_TO_BYTE(t1);

RETURN;

END_FUNCTION

// ---- Object/UDP/DataDecoder.TcPOU
(*
	This class is responsible for extracting
	metadata from a UDP packet. 
*)
FUNCTION_BLOCK DataDecoder
VAR
	
	_Udp						: ITF_UdpConnection;
	_UdpReceiveBuffer			: REFERENCE TO ARRAY [0..TCPADS_MAXUDP_BUFFSIZE - 1] OF BYTE;
	_LastCheckedIndex			: UDINT;
	_PacketsReceived			: ULINT;
	
END_VAR

VAR CONSTANT
	
	_StartDelimiter1			: BYTE := GVL_Udp.StartDelimiter1;
	_StartDelimiter2			: BYTE := GVL_Udp.StartDelimiter2;
	_EndDelimiter1				: BYTE := GVL_Udp.EndDelimiter1;
	_EndDelimiter2				: BYTE := GVL_Udp.EndDelimiter2;
	_PacketTypePosition			: BYTE := GVL_Udp.PacketTypePosition;
	
END_VAR

METHOD ClearBufferAtLocation : BOOL
VAR_INPUT
	PacketAddress			: PVOID;
	PacketLength			: UINT;
END_VAR
VAR
	i	: UDINT;
END_VAR

IF MEMSET(PacketAddress, 0, PacketLength) > 0 THEN

	ClearBufferAtLocation := TRUE;
	
ELSE
	
	ClearBufferAtLocation := FALSE;
	
END_IF

RETURN;
END_METHOD

METHOD CreateMetadataUpdate : EspPacketHeader
VAR_INPUT
END_VAR

MEMCPY(ADR(CreateMetadataUpdate), ADR(_UdpReceiveBuffer[0]), 48);

RETURN;
END_METHOD

//FB_Init is always available implicitly and it is used primarily for initialization.
//The return value is not evaluated. For a specific influence, you can also declare the
//methods explicitly and provide additional code there with the standard initialization
//code. You can evaluate the return value.
METHOD FB_Init: BOOL
VAR_INPUT
    bInitRetains: BOOL; // TRUE: the retain variables are initialized (reset warm / reset cold)
    bInCopyCode: BOOL;  // TRUE: the instance will be copied to the copy code afterward (online change)   
	UdpSocket	: ITF_UdpConnection;
	EspList		: ITF_LinkedList;
END_VAR
_Udp := UdpSocket;
_UdpReceiveBuffer REF= _Udp.ReceiveBufferReference;
END_METHOD

METHOD GetPacketHeader : EspPacketHeader
VAR_INPUT
END_VAR
MEMCPY(ADR(GetPacketHeader), ADR(_UdpReceiveBuffer[0]), 48);
END_METHOD

METHOD GetPacketUID : ULINT
VAR_INPUT
END_VAR
MEMCPY(ADR(GetPacketUID), ADR(_UdpReceiveBuffer[8]), 8);
END_METHOD

METHOD TryFindPacketInBuffer : HRESULT
VAR_INPUT
	PacketType				: REFERENCE TO BYTE;
	PacketAddress			: REFERENCE TO PVOID;
	PacketLength			: REFERENCE TO UINT;
	DataLength				: REFERENCE TO UINT;
END_VAR
VAR
	i						: UDINT;
	Good					: BOOL;
END_VAR
TryFindPacketInBuffer := S_PENDING;

IF NOT _Udp.IsConnected() OR ADR(_UdpReceiveBuffer) = 0 THEN
	
	RETURN;

END_IF

FOR i := _LastCheckedIndex TO TCPADS_MAXUDP_BUFFSIZE - 1 BY 1 DO
	
	IF _UdpReceiveBuffer[i] = _StartDelimiter1 AND_THEN _UdpReceiveBuffer[i + 1] = _StartDelimiter2 THEN
					
		PacketType := _UdpReceiveBuffer[i + _PacketTypePosition];
		
		PacketAddress := ADR(_UdpReceiveBuffer[i]);
		
		DataLength := BytesToUint(_UdpReceiveBuffer[i + 2], _UdpReceiveBuffer[i + 3]);
		
		PacketLength := 48 + DataLength + 2;
		
		IF DataLength = 0 OR PacketType = 0 THEN
			
			TryFindPacketInBuffer := -1;
					
		ELSIF _UdpReceiveBuffer[i + 48 + DataLength] <> _EndDelimiter1 OR _UdpReceiveBuffer[i + 48 + DataLength + 1] <> _EndDelimiter2 THEN
			
			TryFindPacketInBuffer := S_PENDING;
			
		ELSE
			
			_PacketsReceived := _PacketsReceived + 1;
			
			Good := TRUE;
			
		END_IF
		
		EXIT;
					
	END_IF

END_FOR

IF _LastCheckedIndex > TCPADS_MAXUDP_BUFFSIZE - 1 THEN
	
	_LastCheckedIndex := 0;
	
ELSE
	
	_LastCheckedIndex := i;

END_IF

IF Good THEN
	
	TryFindPacketInBuffer := S_OK;
	
ELSE
	
	TryFindPacketInBuffer := -1;

END_IF

RETURN;
END_METHOD

END_FUNCTION_BLOCK

// ---- Functions/BytesToUint.TcPOU
FUNCTION BytesToUint : UINT
VAR_INPUT
	b1	: BYTE;
	b2	: BYTE;
END_VAR

BytesToUint := TO_UINT(b2) 
			+ TO_UINT(b1) * 256;

END_FUNCTION

// ---- Object/ESP/UpdaterRegistry.TcPOU
FUNCTION_BLOCK UpdaterRegistry IMPLEMENTS ITF_UpdaterRegistry
VAR
	Entries					: ARRAY [0..255] OF UpdaterEntry;
	EntryCount				: BYTE := 0;
	
	RegisterOkCount         : UDINT;
    RegisterDuplicateCount  : UDINT;
    RegisterTableFullCount  : UDINT;
    ResolveMissExactCount   : UDINT;
    ResolveMissTypeCount    : UDINT;
END_VAR

METHOD Reset : BOOL
VAR
	i		: BYTE;
END_VAR

FOR i := 0 TO EntryCount BY 1 DO
	
	Entries[i].TypeID := 0;
	Entries[i].Version := 0;
	Entries[i].Updater := 0;

END_FOR

EntryCount := 0;
RegisterOkCount := 0;
RegisterDuplicateCount := 0;
RegisterTableFullCount := 0;
ResolveMissExactCount := 0;
ResolveMissTypeCount := 0;
END_METHOD

METHOD ResolveUpdater : ITF_Updater
VAR_INPUT
	TypeID	: BYTE;
	Version	: BYTE;
END_VAR
VAR
	i		: BYTE;
END_VAR
ResolveUpdater := 0;

// Exact match (type + version)
FOR i := 0 TO EntryCount - 1 DO
	
    IF (Entries[i].TypeID = TypeID) AND (Entries[i].Version = Version) THEN
		
        ResolveUpdater := Entries[i].Updater;
		
        RETURN;
		
    END_IF
	
END_FOR


ResolveMissExactCount := ResolveMissExactCount + 1;

// Fallback: any entry with same type (e.g. default version)
FOR i := 0 TO EntryCount - 1 DO
	
    IF Entries[i].TypeID = TypeID THEN
		
        ResolveUpdater := Entries[i].Updater;
		
        RETURN;
		
    END_IF
	
END_FOR

ResolveMissTypeCount := ResolveMissTypeCount + 1;

RETURN;
END_METHOD

METHOD TryRegister : HRESULT
VAR_INPUT
	Updater	: ITF_Updater;
END_VAR
VAR
    i       : BYTE;
    TypeId  : BYTE;
    Version : BYTE;
END_VAR
TryRegister := S_PENDING;

IF Updater = 0 THEN
	
	TryRegister := -1;	

    RETURN;
	
END_IF

IF EntryCount = 255 THEN
	
    RegisterTableFullCount := RegisterTableFullCount + 1;
	
	TryRegister := -2;
	
    RETURN;
	
END_IF

TypeId  := Updater.GetTypeID();
Version := Updater.GetVersion();

FOR i := 0 TO EntryCount DO

    IF (Entries[i].TypeID = TypeId) AND (Entries[i].Version = Version) THEN
		
        RegisterDuplicateCount := RegisterDuplicateCount + 1;
		
		TryRegister := -3;
		
        RETURN;
    
	END_IF
	
END_FOR

Entries[EntryCount].TypeID  := TypeId;
Entries[EntryCount].Version := Version;
Entries[EntryCount].Updater := Updater;
EntryCount := EntryCount + 1;

RegisterOkCount := RegisterOkCount + 1;

TryRegister := S_OK;

RETURN;
END_METHOD

END_FUNCTION_BLOCK

// ---- Object/ESP/Updater_TestPacket.TcPOU
FUNCTION_BLOCK Updater_TestPacket IMPLEMENTS ITF_Updater
VAR CONSTANT
    PacketID  				: BYTE := 1;
    PacketVersion 			: BYTE := 1;
	PacketSize				: BYTE := 66;
END_VAR
VAR
	TempBuffer				: ARRAY [0..PacketSize - 1] OF BYTE;	

	ApplyOkCount            : UDINT;
    ApplyLengthErrorCount   : UDINT;
    ApplyBufferTooSmall     : UDINT;
END_VAR

METHOD GetTypeID : BYTE
GetTypeID := PacketID;
END_METHOD

METHOD GetVersion : BYTE
GetVersion := PacketVersion;
END_METHOD

METHOD TryApplyPayload : HRESULT
VAR_INPUT
	PacketAddress	: PVOID;
	PacketLength	: UINT;
	EspHost			: ITF_EspHost;
END_VAR
VAR
    BufferAddress : PVOID;
    BufferSize    : UDINT;
END_VAR
TryApplyPayload := S_PENDING;

IF PacketLength <> PacketSize THEN
	
    ApplyLengthErrorCount := ApplyLengthErrorCount + 1;
	
	TryApplyPayload := -1;
	
	RETURN;
	
END_IF

IF NOT EspHost.GetDataBuffer(BufferAddress, BufferSize) THEN
	
	TryApplyPayload := -2;

    RETURN;
	
END_IF

IF PacketLength > BufferSize THEN
	
    ApplyBufferTooSmall := ApplyBufferTooSmall + 1;
	
    TryApplyPayload := -3;
    
	RETURN;

END_IF



MEMCPY(BufferAddress, PacketAddress, PacketLength);

ApplyOkCount := ApplyOkCount + 1;

TryApplyPayload := S_OK;          // success

RETURN;
END_METHOD

METHOD TryGetContents : HRESULT
VAR_INPUT
	Host	: ITF_EspHost;
	Content	: REFERENCE TO STRING(1024);
END_VAR
VAR
    BufferAddress 	: PVOID;
    BufferSize   	: UDINT;
	td9 			: ULINT;
END_VAR
TryGetContents := S_PENDING;

Content := '{"Error" : "No_Data_Available"}';

IF NOT Host.GetDataBuffer(BufferAddress, BufferSize) THEN

	TryGetContents := -1;	

    RETURN;
	
END_IF

IF MEMCPY(ADR(TempBuffer), BufferAddress, BufferSize) <= 0 THEN
	
	TryGetContents := -2;
	
	RETURN;

END_IF

Content := '';

Content := CONCAT(Content, '{"Test_Data_1" : ');
Content := CONCAT(Content, TO_STRING(TempBuffer[48]));
Content := CONCAT(Content, ', "Test_Data_2" : ');
Content := CONCAT(Content, TO_STRING(TempBuffer[49]));
Content := CONCAT(Content, ', "Test_Data_3" : ');
Content := CONCAT(Content, TO_STRING(TempBuffer[50]));
Content := CONCAT(Content, ', "Test_Data_4" : ');
Content := CONCAT(Content, TO_STRING(TempBuffer[51]));
Content := CONCAT(Content, ', "Test_Data_5" : ');
Content := CONCAT(Content, TO_STRING(TempBuffer[52]));
Content := CONCAT(Content, ', "Test_Data_6" : ');
Content := CONCAT(Content, TO_STRING(TempBuffer[53]));
Content := CONCAT(Content, ', "Test_Data_7" : ');
Content := CONCAT(Content, TO_STRING(TempBuffer[54]));
Content := CONCAT(Content, ', "Test_Data_8" : ');
Content := CONCAT(Content, TO_STRING(TempBuffer[55]));

td9 := (TempBuffer[56]);
td9 := SHL(td9, 8) OR (TempBuffer[57]);
td9 := SHL(td9, 8) OR (TempBuffer[58]);
td9 := SHL(td9, 8) OR (TempBuffer[59]);
td9 := SHL(td9, 8) OR (TempBuffer[60]);
td9 := SHL(td9, 8) OR (TempBuffer[61]);
td9 := SHL(td9, 8) OR (TempBuffer[62]);
td9 := SHL(td9, 8) OR (TempBuffer[63]);

Content := CONCAT(Content, ', "Test_Data_9" : ');
Content := CONCAT(Content, TO_STRING(td9));
Content := CONCAT(Content, '}');

TryGetContents := S_OK;

RETURN;
END_METHOD

{warning 'Add method implementation '}
METHOD TrySendInstruction : HRESULT
END_METHOD

END_FUNCTION_BLOCK

// ---- Object/ESP/EspHost.TcPOU
{attribute 'enable_dynamic_creation'}
FUNCTION_BLOCK EspHost IMPLEMENTS ITF_EspHost, ITF_Node
VAR
	
	// Node information
	_LastNode					: ITF_Node;
	_NextNode					: ITF_Node;
	_PositionInList				: UINT;
	
	
	
	// ESP information
	_Data						: EspPacketHeader;
	_PacketsReceivedCount		: ULINT;
	_LastReceivedTimestamp		: ULINT;
	_DataBuffer					: ARRAY [0..511] OF BYTE;
	
END_VAR

METHOD CyclicUpdate : BOOL
VAR_INPUT
END_VAR
END_METHOD

METHOD GetDataBuffer : BOOL
VAR_INPUT
	Address	: REFERENCE TO PVOID;
	Size	: REFERENCE TO UDINT;
END_VAR
Address := ADR(_DataBuffer);
Size := SIZEOF(_DataBuffer);

GetDataBuffer := TRUE;
END_METHOD

METHOD GetLastNode : ITF_Node
GetLastNode := _LastNode;

RETURN;
END_METHOD

METHOD GetMetadata : EspPacketHeader
VAR_INPUT
END_VAR
GetMetadata := _Data;
END_METHOD

METHOD GetMyPointer : PVOID
GetMyPointer := ADR(THIS^);
END_METHOD

METHOD GetNextNode : ITF_Node
GetNextNode := _NextNode;

RETURN;
END_METHOD

{warning 'Add method implementation '}
METHOD GetPacketToSend : BOOL
VAR_INPUT
	Address	: REFERENCE TO PVOID;
	Size	: REFERENCE TO UDINT;
END_VAR
GetPacketToSend := FALSE;
END_METHOD

METHOD GetPositionInList : UINT
GetPositionInList := _PositionInList;

RETURN;
END_METHOD

METHOD SetEspType : BOOL
VAR_INPUT
	EspType	: BYTE;
END_VAR
IF _Data.EspType = 0 THEN
	
	_Data.EspType := EspType;
	
	SetEspType := TRUE;

END_IF

RETURN;
END_METHOD

METHOD SetLastNode : BOOL
VAR_INPUT
	Node	: ITF_Node;
END_VAR
_LastNode := Node;

SetLastNode := TRUE;

RETURN;
END_METHOD

METHOD SetNextNode : BOOL
VAR_INPUT
	Node	: ITF_Node;
END_VAR
_NextNode := Node;

SetNextNode := TRUE;

RETURN;
END_METHOD

METHOD SetPositionInList : BOOL
VAR_INPUT
	Index	: UINT;
END_VAR
_PositionInList := Index;

SetPositionInList := TRUE;

RETURN;
END_METHOD

METHOD SetUID : BOOL
VAR_INPUT
	UID	: ULINT;
END_VAR
IF _Data.SlaveUid = 0 THEN
	
	_Data.SlaveUid := UID;
	
	SetUID := TRUE;

END_IF

RETURN;
END_METHOD

METHOD UpdateMetadata : BOOL
VAR_INPUT
	Data	: EspPacketHeader;
END_VAR
IF MEMCPY(ADR(_Data), ADR(Data), 48) = 48 THEN
	
	_PacketsReceivedCount := _PacketsReceivedCount + 1;	

	_LastReceivedTimestamp := F_GetSystemTime();

	UpdateMetadata := TRUE;
	
ELSE
	
	UpdateMetadata := FALSE;

END_IF


// IF Data.SendersTimestamp <> 0 THEN
// 	
// 	_Data.SendersTimestamp := Data.SendersTimestamp;
// 
// END_IF
// 
// IF Data.TimeDifference <> 0 THEN
// 	
// 	_Data.TimeDifference := Data.TimeDifference;
// 
// END_IF
// 
// UpdateMetadata := TRUE;
// 
// _PacketsReceivedCount := _PacketsReceivedCount + 1;
// 
// RETURN;
END_METHOD

END_FUNCTION_BLOCK

// ---- Functions/HeaderEndianSwap.TcPOU
FUNCTION HeaderEndianSwap : EspPacketHeader
VAR_INPUT
	In	: EspPacketHeader;
END_VAR
VAR
END_VAR

In.StartDelimiter        := BE16_TO_HOST(In.StartDelimiter);
In.PayloadSize           := BE16_TO_HOST(In.PayloadSize);
In.SlaveUid              := BE64_TO_HOSTEX(In.SlaveUid);
In.MessageCounter        := BE64_TO_HOSTEX(In.MessageCounter);
In.SendersTimestamp      := BE64_TO_HOSTEX(In.SendersTimestamp);
In.TimeDifference        := BE32_TO_HOST(In.TimeDifference);
In.CRC32                 := BE32_TO_HOST(In.CRC32);

HeaderEndianSwap := In;

END_FUNCTION

// ---- POUs/EnergyCalculator.TcPOU
FUNCTION_BLOCK EnergyCalculator
VAR_INPUT
	Voltage							: LREAL;
	Current							: LREAL;
END_VAR
VAR_OUTPUT	
	PowerConsumptionAverageW		: LREAL;
	EnergyConsumptionTotalJ			: LREAL;
	EnergyConsumptionTotalkWh		: LREAL;
	EnergyConsumptionCostPence		: LREAL;
END_VAR
VAR
	Initialized						: BOOL;
	TaskIndex						: DINT;
	TaskTimeS						: REAL;
	CyclesExecuted					: ULINT;
	PowerConsumptionW				: LREAL;
	PowerConsumptionThisCycleJ		: LREAL;
	TimeAliveS						: LREAL;
END_VAR
VAR CONSTANT
	EnergyPricePence				: REAL := 26.35;
END_VAR


CyclesExecuted := CyclesExecuted + 1;

IF NOT Initialized THEN
	
	TaskIndex := GETCURTASKINDEXEX();
	
	TaskTimeS := _TaskInfo[TaskIndex].CycleTime / 10000000.0;
	
	Initialized := TRUE;

END_IF

PowerConsumptionW := Voltage * Current;

PowerConsumptionThisCycleJ := PowerConsumptionW * TaskTimeS;

EnergyConsumptionTotalJ := EnergyConsumptionTotalJ + PowerConsumptionThisCycleJ;

EnergyConsumptionTotalkWh := EnergyConsumptionTotalJ / 3600000.0;

TimeAliveS := CyclesExecuted * TaskTimeS;

IF TimeAliveS <> 0 THEN
	
	PowerConsumptionAverageW := EnergyConsumptionTotalJ / TimeAliveS;

END_IF

EnergyConsumptionCostPence := EnergyConsumptionTotalkWh * EnergyPricePence;

END_FUNCTION_BLOCK

// ---- POUs/MessageBuffer.TcPOU
FUNCTION_BLOCK MessageBuffer
VAR
	Buffer	: ARRAY [0..1023] OF STRING(1024);
END_VAR

METHOD AddData : BOOL
VAR_INPUT
	Data	: STRING(1024);
END_VAR
VAR
	i		: UINT;
END_VAR
IF Data = '' THEN

	RETURN;	

END_IF

FOR i := 1023 TO 1 BY -1 DO
	
	Buffer[i] := Buffer[i - 1];

END_FOR

Buffer[0] := Data;

AddData := TRUE;
END_METHOD

END_FUNCTION_BLOCK

// ---- POUs/Utility.TcPOU
PROGRAM Utility
VAR
	LedStrip						: RgbController;
	Red								: BOOL := FALSE;
	Green							: BOOL := TRUE;
	Blue							: BOOL := FALSE;
	
	EL9227Ch1						: MDP5001_922_DEB3C1CF;
	EL9227Ch2						: MDP5001_922_DEB3C1CF;
	
	EnergyCalculator				: EnergyCalculator;
	EnergyConsumptionCostPence		: LREAL;
	
END_VAR


EnergyCalculator
(
	Voltage						:= EL9227Ch1.MDP5001_922_Input.MDP5001_922_Voltage_In / 10.0, 
	Current						:= EL9227Ch1.MDP5001_922_Input.MDP5001_922_Current / 100.0,
	PowerConsumptionAverageW	=> ,
	EnergyConsumptionTotalJ		=> , 
	EnergyConsumptionTotalkWh	=> ,
	EnergyConsumptionCostPence	=> EnergyConsumptionCostPence
);

LedStrip.SetCustom(Red, Green, Blue);

END_PROGRAM

// ---- Tests/TestNode.TcPOU
{attribute 'enable_dynamic_creation'}
FUNCTION_BLOCK TestNode IMPLEMENTS ITF_Node
VAR
	_next : ITF_Node;
    _prev : ITF_Node;
    _pos  : UINT;
END_VAR

METHOD GetLastNode : ITF_Node
GetLastNode := _prev;
END_METHOD

METHOD GetMyPointer : PVOID
GetMyPointer := ADR(THIS^);
END_METHOD

METHOD GetNextNode : ITF_Node
GetNextNode := _next;
END_METHOD

METHOD GetPositionInList : UINT
GetPositionInList := _pos;
END_METHOD

METHOD SetLastNode : BOOL
VAR_INPUT
	Node	: ITF_Node;
END_VAR
_prev := Node; 

SetLastNode := TRUE;
END_METHOD

METHOD SetNextNode : BOOL
VAR_INPUT
	Node	: ITF_Node;
END_VAR
_next := Node; 

SetNextNode := TRUE;
END_METHOD

METHOD SetPositionInList : BOOL
VAR_INPUT
	Index	: UINT;
END_VAR
_pos := Index; 

SetPositionInList := TRUE;
END_METHOD

END_FUNCTION_BLOCK

// ---- Tests/TestNodeFactory.TcPOU
FUNCTION_BLOCK TestNodeFactory IMPLEMENTS ITF_NodeFactory
VAR
	CreatedCount : UDINT;
    DeletedCount : UDINT;
END_VAR

METHOD CreateNode : ITF_Node
VAR
	p : POINTER TO TestNode;
END_VAR
p := __NEW(TestNode);
IF p <> 0 THEN
    CreatedCount := CreatedCount + 1;
    CreateNode := p^;   // return as ITF_Node
END_IF
END_METHOD

METHOD DestroyNode : BOOL
VAR_INPUT
	Ptr	: PVOID;
END_VAR
VAR 
	p : POINTER TO TestNode; 
END_VAR
p := Ptr;
IF p <> 0 THEN
    __DELETE(p);
    DeletedCount := DeletedCount + 1;
    DestroyNode := TRUE;
END_IF
END_METHOD

METHOD DoesCreateEqualDestroy : BOOL
VAR_INPUT
END_VAR
IF CreatedCount = DeletedCount THEN

	DoesCreateEqualDestroy := TRUE;

ELSE

	DoesCreateEqualDestroy := FALSE;	

END_IF
END_METHOD

END_FUNCTION_BLOCK

// ---- Tests/Tests_ListAndFactory.TcPOU
PROGRAM Tests_ListAndFactory
VAR
    T 			: TestHarness;
	f1			: TestNodeFactory;
	f2			: EspNodeFactory;
	Factory 	: ITF_NodeFactory := f2;
	List		: List(Factory);
    UUT 		: ITF_LinkedList := List;          
    Done	 	: BOOL := FALSE;

    ok 			: BOOL;
    len 		: UINT;

	p1, p2, i		: UINT;
    n1, n2, n3, tmp : ITF_Node;     
END_VAR

IF NOT Done THEN

	// --- Fresh harness ----------------------------------------------------------------------------------------------------
	
	T.Clear();



	// --- Delete on empty --------------------------------------------------------------------------------------------------
	
	ok := UUT.DestroyNode(1);							T.AssertTrue(NOT ok, 'delete on empty returns FALSE');



	// --- Create and delete node -------------------------------------------------------------------------------------------
	
	ok := UUT.CreateNode();								T.AssertTrue(ok, 'CreateNode #1 ok');
	len := UUT.GetListLength(); 						T.AssertTrue(len = 1, 'len=1 after first create');
	n1 := UUT.GetNode(Index := 1); 						T.AssertTrue(n1 <> 0, 'GetNode(1) not null');

	ok := UUT.DestroyNode(Index := 1); 					T.AssertTrue(ok, 'delete index 1 ok');
	len := UUT.GetListLength(); 						T.AssertTrue(len = 0, 'len=0 after delete last');
	tmp := UUT.GetNode(Index := 1);						T.AssertTrue(tmp = 0, 'GetNode(1) null after delete');



	// --- Create three nodes and check pointers ----------------------------------------------------------------------------
	
	ok := UUT.CreateNode();								T.AssertTrue(ok, 'CreateNode #1 ok');
	ok := UUT.CreateNode();								T.AssertTrue(ok, 'CreateNode #2 ok');
	ok := UUT.CreateNode();								T.AssertTrue(ok, 'CreateNode #3 ok');
	len := UUT.GetListLength();							T.AssertTrue(len = 3, 'len=3 after three creates');

	n1 := UUT.GetNode(1);
	n2 := UUT.GetNode(2); 
	n3 := UUT.GetNode(3);								T.AssertTrue(n1 <> 0 AND n2 <> 0 AND n3 <> 0, 'nodes 1..3 exist');
	
	tmp := n1.GetLastNode();							T.AssertTrue(tmp = 0, '1.prev = NULL');
	tmp := n1.GetNextNode();							T.AssertTrue(tmp = n2, '1.next = 2');
	tmp := n2.GetLastNode();							T.AssertTrue(tmp = n1, '2.prev = 1');
	tmp := n2.GetNextNode();							T.AssertTrue(tmp = n3, '2.next = 3');
	tmp := n3.GetLastNode();							T.AssertTrue(tmp = n2, '3.prev = 2');
	tmp := n3.GetNextNode();							T.AssertTrue(tmp = 0, '3.next = NULL');
	
	len := UUT.GetListLength();							T.AssertTrue(len = 3, 'pre: len=3');
	
	
	
	// --- Test invalid nodes ------------------------------------------------------------------------------------------
	
	tmp := UUT.GetNode(0);								T.AssertTrue(tmp = 0, 'GetNode(0)=0');
	tmp := UUT.GetNode(-1);								T.AssertTrue(tmp = 0, 'GetNode(-1)=0');
	tmp := UUT.GetNode(4);								T.AssertTrue(tmp = 0, 'GetNode(4)=0');
	
	
	ok := UUT.DestroyNode(0);							T.AssertTrue(NOT ok, 'delete on 0 returns FALSE');
	ok := UUT.DestroyNode(-1);							T.AssertTrue(NOT ok, 'delete on negative returns FALSE');
	ok := UUT.DestroyNode(4);							T.AssertTrue(NOT ok, 'delete on 4 (outside list) returns FALSE');



	// --- Delete middle (index 2) ------------------------------------------------------------------------------------------
	
	ok := UUT.DestroyNode(Index := 2);					T.AssertTrue(ok, 'delete middle ok');
	len := UUT.GetListLength();							T.AssertTrue(len = 2, 'len=2 after middle delete');

	n1 := UUT.GetNode(1);
	n2 := UUT.GetNode(2);
	tmp := n1.GetNextNode();							T.AssertTrue(tmp = n2, 'after delete: 1.next = 2');
	tmp := n2.GetLastNode();							T.AssertTrue(tmp = n1, 'after delete: 2.prev = 1');

	p1 := n1.GetPositionInList();						T.AssertTrue(p1 = 1, 'pos(1)=1 after delete');
	p2 := n2.GetPositionInList();						T.AssertTrue(p2 = 2, 'pos(2)=2 after delete');
	


	// --- Delete head on 2-node list ---------------------------------------------------------------------------------------
	
	ok := UUT.DestroyNode(Index := 1);					T.AssertTrue(ok, 'delete head ok');
	len := UUT.GetListLength();							T.AssertTrue(len = 1, 'len=1 after delete head');

	n1 := UUT.GetNode(1);								T.AssertTrue(n1 <> 0, 'single node exists');
	tmp := n1.GetLastNode();							T.AssertTrue(tmp = 0, 'single.prev = 0');
	tmp := n1.GetNextNode();							T.AssertTrue(tmp = 0, 'single.next = 0');
	p1 := n1.GetPositionInList();						T.AssertTrue(p1 = 1, 'single pos=1');   



	// --- Delete last remaining node ---------------------------------------------------------------------------------------
	
	ok := UUT.DestroyNode(Index := 1);					T.AssertTrue(ok, 'delete last ok');
	len := UUT.GetListLength();							T.AssertTrue(len = 0, 'len=0 at end');
	tmp := UUT.GetNode(1);								T.AssertTrue(tmp = 0, 'no nodes remain');
	
	
	
	// --- Create list of 3 and destroy by tails ----------------------------------------------------------------------------
	
	UUT.CreateNode(); 
	UUT.CreateNode(); 
	UUT.CreateNode();
	ok := UUT.DestroyNode(3);							T.AssertTrue(ok, 'delete tail ok');
	len := UUT.GetListLength();							T.AssertTrue(len = 2, 'len=2 after tail delete');

	n1 := UUT.GetNode(1); 
	n2 := UUT.GetNode(2);
	tmp := n1.GetNextNode();							T.AssertTrue(tmp = n2, '1.next=2 after tail delete');
	tmp := n2.GetNextNode();							T.AssertTrue(tmp = 0, 'new tail.next=0');
	ok := UUT.DestroyNode(3);							T.AssertTrue(NOT ok, 'do not delete null pointer ok');
	ok := UUT.DestroyNode(2);							T.AssertTrue(ok, 'delete pos=2');
	ok := UUT.DestroyNode(1);							T.AssertTrue(ok, 'delete pos=1');



	// --- Create 100 entries -----------------------------------------------------------------------------------------------
	
	FOR i := 1 TO 100 BY 1 DO
		UUT.CreateNode();
	END_FOR
	len := UUT.GetListLength();							T.AssertTrue(len = 100, 'len=100 after FOR loop creation');



	// --- Destroy 100 entries by head --------------------------------------------------------------------------------------
	
	FOR i := 1 TO 100 BY 1 DO
		UUT.DestroyNode(1);
	END_FOR
	len := UUT.GetListLength();							T.AssertTrue(len = 0, 'len=0 after FOR loop destruction');



	// --- End --------------------------------------------------------------------------------------------------------------

	Done := TRUE; 
	
	
	
END_IF

END_PROGRAM

// ---- Tests/Tests_Udp.TcPOU
PROGRAM Tests_Udp
VAR
	T 			: TestHarness;
	f1			: UdpWindowsSocket('192.168.1.227', 10050);
	f2			: UdpRealtimeSocket(10050);
	UUT1		: ITF_UdpConnection := f2;  
	Cyclic		: ITF_Cyclic := f1;
	ip			: T_IPv4Addr := '192.168.0.2';     
	port		: UINT := 10050;
	SomeData	: STRING := 'Hello World';
	
	 
    Done	 	: BOOL := FALSE;
	State		: BYTE;
	Iterations	: ULINT;
    ok 			: BOOL;
    len 		: UINT;
	hr			: HRESULT;
	p1, p2, i		: UINT;  
END_VAR

Cyclic.CyclicUpdate();


IF NOT Done THEN

	CASE State OF
		
		
		
		0:
		
			// --- Fresh harness ----------------------------------------------------------------------------------------------------
		
			T.Clear();


		
			// --- Test connection and flags BEFORE CONNECTED -----------------------------------------------------------------------
	
			ok := UUT1.IsConnected();											T.AssertTrue(NOT ok, 'IsConnected before connected returns FALSE');
			ok := UUT1.IsSending();												T.AssertTrue(NOT ok, 'IsSending before connected returns FALSE');
			State := 1;
			
			
			
		1:
		
			// --- Test send BEFORE CONNECTED ---------------------------------------------------------------------------------------
		
			hr := UUT1.TrySendData(ip,port,ADR(SomeData),SIZEOF(SomeData));		IF hr <> S_PENDING THEN T.AssertTrue(hr < 0, 'Failed to send data'); END_IF
			IF hr <> S_PENDING THEN
				State := 2;
			END_IF
		
		
		
		2:
		
			// --- Open socket for UDP (does not require external packet-sender) ----------------------------------------------------
			
			hr := UUT1.TryOpenConnection();										IF hr <> S_PENDING THEN T.AssertTrue(hr = S_OK, 'UDP socket open'); END_IF
			IF hr <> S_PENDING THEN
				State := 3;
			END_IF
			
		
		
		3:
		
			// --- Test connection AFTER CONNECTED ----------------------------------------------------------------------------------
	
			ok := UUT1.IsConnected();											T.AssertTrue(ok, 'IsConnected after connected returns TRUE');
			State := 4;
			
			
			
		4:
		
			// --- Test send AFTER CONNECTED ----------------------------------------------------------------------------------------
		
			hr := UUT1.TrySendData(ip,port,ADR(SomeData),SIZEOF(SomeData));		IF hr <> S_PENDING THEN T.AssertTrue(hr = S_OK, 'Successfully send data'); END_IF
			IF hr <> S_PENDING THEN
				State := 5;
			END_IF
			
			
			
		5:
			
			// --- Close socket for UDP (does not require external packet-sender) ---------------------------------------------------
			
			hr := UUT1.TryCloseConnection();									IF hr <> S_PENDING THEN T.AssertTrue(hr = S_OK, 'UDP socket closed'); END_IF
			IF hr = S_OK THEN
				State := 6;
			END_IF
			
			State := 6;
			
			
			
		6:
		
			// --- Test connection and flags AFTER DISCONNECT -----------------------------------------------------------------------
	
			ok := UUT1.IsConnected();											T.AssertTrue(NOT ok, 'IsConnected before connected returns FALSE');
			ok := UUT1.IsSending();												T.AssertTrue(NOT ok, 'IsSending before connected returns FALSE');
			State := 7;
		
		
		
		7:
		
			// --- Test send AFTER DISCONNECTED -------------------------------------------------------------------------------------
		
			hr := UUT1.TrySendData(ip,port,ADR(SomeData),SIZEOF(SomeData));		IF hr <> S_PENDING THEN T.AssertTrue(hr < 0, 'Failed to send data'); END_IF
			IF hr <> S_PENDING THEN
				State := 8;
			END_IF
			
		
		
		8:
		
			Done := TRUE;
			Iterations := Iterations + 1;
			State := 0; 
	
	
	
	END_CASE
		
END_IF

END_PROGRAM
